Fanuc KAREL source: NC0025.KL

-- PROVISIONAL review KL for V940-1; original PC SHA256 ba92fa3185c43d2d683dfe26da5e16b005cd35c7f00b5a7ca1ab613ea7ccbf1d
-- Incomplete behavior may be omitted. Consult companion uncertainty JSON. Do not deploy.
PROGRAM NC0025
%NOLOCKGROUP
-- UNRESOLVED_LOCAL_POOL 1 cells at code offset 3; source declarations unknown
-- DIRECT_LOCAL_WORD_ACCESS alone does not prove INTEGER, REAL, or BOOLEAN
BEGIN
  -- UNRESOLVED_PC offsets 0-8; opcodes 2B,2C,7B
  -- UNRESOLVED_PC offsets 13-20; opcodes 9D,23
  -- UNRESOLVED_PC offsets 25-42; opcodes 21,40,41,42
  -- UNRESOLVED_PC offsets 47-64; opcodes 21,40,41,42
  -- UNRESOLVED_PC offsets 69-86; opcodes 21,40,41,42
  -- UNRESOLVED_PC offsets 91-108; opcodes 21,40,41,42
  -- UNRESOLVED_PC offsets 113-130; opcodes 21,40,41,42
  -- UNRESOLVED_PC offsets 135-165; opcodes 21,9D,52,23,7A,40,41,42
  -- UNRESOLVED_PC offsets 170-194; opcodes 21,2E,52,23,7A,43
  -- UNRESOLVED_PC offsets 199-217; opcodes 21,2E,52,23
  -- UNRESOLVED_PC offsets 222-238; opcodes 7A,40,41,42
  -- UNRESOLVED_PC offsets 243-267; opcodes 21,2E,52,23,7A,43
  -- UNRESOLVED_PC offsets 272-290; opcodes 21,2E,52,23
  -- UNRESOLVED_PC offsets 295-311; opcodes 7A,40,41,42
  -- UNRESOLVED_PC offsets 316-340; opcodes 21,2E,52,23,7A,43
  -- UNRESOLVED_PC offsets 345-363; opcodes 21,2E,52,23
  -- UNRESOLVED_PC offsets 368-384; opcodes 7A,40,41,42
  -- UNRESOLVED_PC offsets 389-413; opcodes 21,2E,52,23,7A,43
  -- UNRESOLVED_PC offsets 418-436; opcodes 21,2E,52,23
  -- UNRESOLVED_PC offsets 441-457; opcodes 7A,40,41,42
  -- UNRESOLVED_PC offsets 462-486; opcodes 21,2E,52,23,7A,43
  -- UNRESOLVED_PC offsets 491-509; opcodes 21,2E,52,23
  -- UNRESOLVED_PC offsets 519-523; opcodes 7F
  -- UNRESOLVED_PC offsets 528-532; opcodes 27,AA
  -- UNRESOLVED_PC offsets 537-541; opcodes 7F
END NC0025
